// SIMATIC S7-200 project (STEP 7-Micro/WIN), CPU 224 REL 01.11

SYMBOL_TABLE USER1
Thuan            I0.0
Nghich           I0.1
Dung             I0.2
Ena              Q0.0
Forr             Q0.1
Rev              Q0.2
T4_              Q0.3
B7               Q0.4
END_SYMBOL_TABLE

ORGANIZATION_BLOCK MAIN:OB1
TITLE=PROGRAM COMMENTS
BEGIN
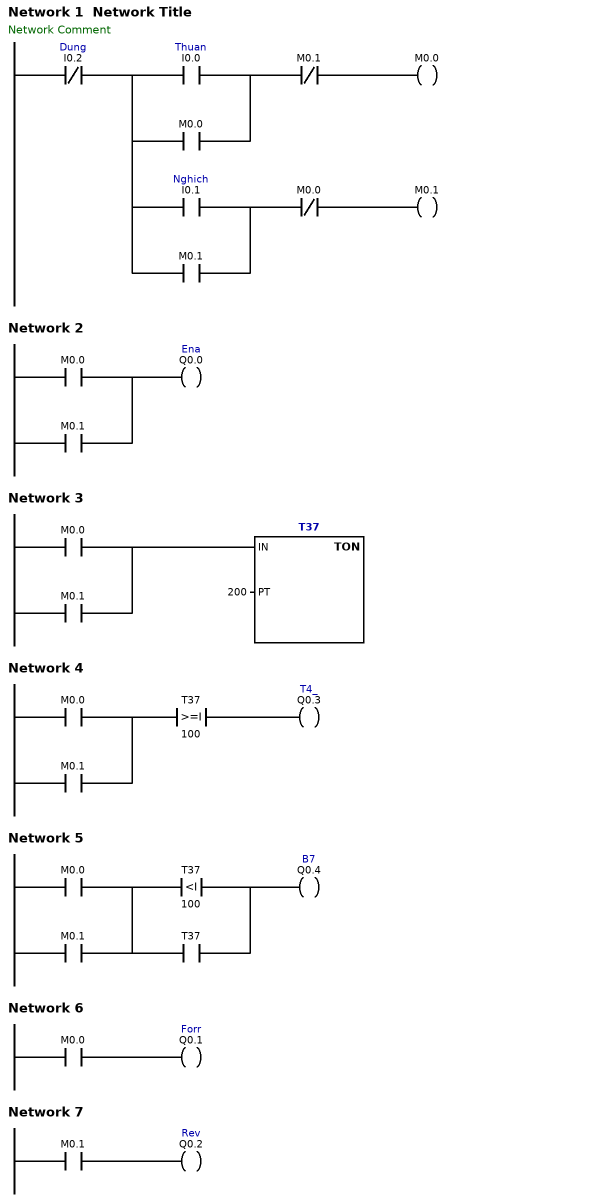
Network 1 // Network Title
// Network Comment
LDN    Dung:I0.2
LPS
LD     Thuan:I0.0
O      M0.0
ALD
AN     M0.1
=      M0.0
LPP
LD     Nghich:I0.1
O      M0.1
ALD
AN     M0.0
=      M0.1
Network 2
LD     M0.0
O      M0.1
=      Ena:Q0.0
Network 3
LD     M0.0
O      M0.1
TON    T37, 200
Network 4
LD     M0.0
O      M0.1
AW>=   T37, 100
=      T4_:Q0.3
Network 5
LD     M0.0
O      M0.1
LDW<   T37, 100
O      T37
ALD
=      B7:Q0.4
Network 6
LD     M0.0
=      Forr:Q0.1
Network 7
LD     M0.1
=      Rev:Q0.2
END_ORGANIZATION_BLOCK
